Staubli VAL3: EXAMPLE.pgx

public program Example()
  local num l_nLine
  local bool l_bBool
  local string l_sString
begin
  cls()
  title("读写文本实例")


  //*********************************************************************
  //新建文本
  gotoxy(0,0)
  put("新建文本HelloVal3.txt")
  nFileID=$fileOpen("Disk://txt/HelloVal3.txt","w")
  if nFileID<0 or nFileID>9
    gotoxy(0,1)
    put("新建打开文件出错！")
    return
  endIf

  //书写文本
  call WriteLine(nFileID,"Hello Val3!",l_bBool)
  if !l_bBool
    gotoxy(0,2)
    put("写入文件出错！")
    return
  endIf

  //关闭文件
  $fileClose(nFileID)

  //*************************************************************************
  //读取文件
  gotoxy(0,0)
  put("读取文本HelloVal3.txt")
  nFileID=$fileOpen("Disk://txt/HelloVal3.txt","r")
  if nFileID<0 or nFileID>9
    gotoxy(0,1)
    put("读取打开文件出错！")
    return
  endIf

  call GetLine(nFileID,l_sString,l_bBool)
  gotoxy(0,2)
  if !l_bBool
    put("读取文件出错！")
    return
  else
    put(l_sString)
  endIf

  //关闭文件
  $fileClose(nFileID)

  //****************************************************************************
  //添加文本
  gotoxy(0,0)
  put("添加文本HelloVal3.txt")
  nFileID=$fileOpen("Disk://txt/HelloVal3.txt","a")
  if nFileID<0 or nFileID>9
    gotoxy(0,1)
    put("添加打开文件出错！")
    return
  endIf

  //书写文本
  call WriteLine(nFileID,"Hello Val3!",l_bBool)
  if !l_bBool
    gotoxy(0,2)
    put("添加写入文件出错！")
    return
  endIf

  //关闭文件
  $fileClose(nFileID)


  //****************************************************************************
  // 删除文本
  gotoxy(0,6)
  if $delete("Disk://txt/HelloVal3.txt")
    put("删除文本成功!")
    return
  else
    put("删除文本失败!")
  endIf

end
